Yaskawa INFORM job: R1_W43-44-A1(80,0))KM-OK.JBI

/JOB
//NAME R1_W43-44-A1(80,0))KM-OK
///FOLDERNAME KRIS-SCIANA
//POS
///NPOS 73,73,0,2,0,0
///TOOL 0
///POSTYPE PULSE
///PULSE
C00000=-135443,-162925,-128835,58859,85380,-57426
C00001=-92446,-155127,-126363,-9824,7934,-58174
C00002=-95529,-35335,-68837,19375,71902,-55615
C00003=-93187,-33344,-64604,18324,69907,-55135
C00004=-92721,-33324,-62151,18250,68383,-55215
C00005=-92468,-33122,-62017,18114,68351,-55131
C00006=-92880,-32499,-63991,18157,69897,-55031
C00007=-84694,-8010,-53588,6240,80947,-57198
C00008=-85014,-7064,-52060,6394,80518,-57316
C00009=-94295,-4530,-48038,22759,83190,-56081
C00010=-78802,-31555,-64347,-3071,67769,-50088
C00011=-78740,-31977,-64165,-3112,67443,-50058
C00012=-84933,-42926,-65553,8148,56142,-50726
C00013=-85694,-44675,-67677,8643,56621,-50981
C00014=-87687,-49011,-72903,9923,57813,-51634
C00015=-99004,-1535,-61632,22381,96772,-38436
C00016=-102646,2603,-65705,33052,95452,-62364
C00017=-97086,-22377,-78433,26069,74095,-68203
C00018=-96393,-22401,-76155,25819,72642,-68318
C00019=-97109,-22798,-76330,26266,72736,-68521
C00020=-97539,-22766,-76077,26544,72724,-68660
C00021=-97679,-22998,-75695,26674,72441,-68771
C00022=-99521,-21962,-80767,27350,76192,-68453
C00023=-70334,1557,-81441,-17401,103237,-40141
C00024=-67843,821,-73813,-18833,98965,-38392
C00025=-100316,3447,-64995,31985,94788,-61866
C00026=-99352,5668,-64520,31595,95249,-61456
C00027=-67843,821,-73813,-18833,98965,-38392
C00028=-85169,3045,-72107,6876,98019,-48310
C00029=-88969,4814,-69933,12844,98216,-50436
C00030=-98274,12123,-60045,27665,97638,-54760
C00031=-89932,6221,-75495,14866,97258,-51043
C00032=-93334,-9371,-63962,22562,99535,9595
C00033=-81626,10879,-49110,8622,108143,9572
C00034=-81231,10229,-48763,8499,107567,9646
C00035=-101964,-23029,-75036,41591,75550,70706
C00036=-102642,-26334,-76142,42122,75049,70241
C00037=-68700,15797,-43598,-6640,106638,27823
C00038=-63261,32591,-26999,-16022,110451,41229
C00039=-64996,36990,-21704,-15609,109207,40852
C00040=-64582,37586,-20939,-15664,109117,40995
C00041=-64496,38242,-20138,-15663,108980,41040
C00042=-64452,38361,-19695,-15647,108783,41080
C00043=-63126,40414,-20326,-16036,110391,41278
C00044=-63319,38327,-23499,-16110,111203,41105
C00045=-43516,29964,-10756,-46242,106248,64597
C00046=-43516,29964,-10756,-46242,106248,64597
C00047=-44396,28590,-11734,-46107,105755,64428
C00048=-43489,29718,-10008,-46103,105848,64806
C00049=-43472,27528,-13134,-46300,106419,64534
C00050=-43936,27041,-10805,-45843,105007,65003
C00051=-43522,29411,-9763,-46025,105613,64905
C00052=-42525,34492,-7112,-46386,106783,64798
C00053=-50383,13985,-41562,-28831,100075,68121
C00054=-64860,2482,-48793,-13393,87629,68164
C00055=-65930,5187,-46476,-12954,87445,67868
C00056=-57792,20564,-34513,-26464,97158,66415
C00057=-62898,8945,-45188,-24852,96370,64962
C00058=-63534,7410,-44996,-24591,95381,64971
C00059=-64227,9067,-43380,-24356,95073,64814
C00060=-63201,10906,-47674,-24936,98605,64395
C00061=-65206,-18847,-70813,-6241,82992,71232
C00062=-69426,-22420,-61359,-4258,75131,70311
C00063=-74955,-30598,-67106,-1464,74288,68599
C00064=-74021,-28518,-73716,-1903,79440,68812
C00065=-70812,-2884,-58486,-3475,83329,69650
C00066=-67265,-11111,-54966,-11415,75263,68927
C00067=-73959,-21777,-63314,-7907,74217,66930
C00068=-72807,-23542,-67362,-8463,75887,67172
C00069=-65188,-31999,-95671,-12172,89534,68158
C00070=-93091,-31999,-95671,-12172,89534,68158
C00071=-92446,-155127,-126363,-9824,7934,-58174
C00072=-92446,-155127,-126363,-9824,7934,84739
BC00000=21010,537295,1075111
BC00001=71,16,1075106
BC00002=15,15,1075175
BC00003=15,15,1075175
BC00004=15,15,1075175
BC00005=15,15,1075175
BC00006=15,15,1075175
BC00007=15,15,1075175
BC00008=15,15,1075175
BC00009=15,15,1075175
BC00010=15,15,1075175
BC00011=15,15,1075175
BC00012=15,15,1075175
BC00013=15,15,1075175
BC00014=15,15,1075175
BC00015=15,15,1006509
BC00016=15,15,928033
BC00017=15,15,898387
BC00018=15,15,898387
BC00019=15,15,898387
BC00020=15,15,898387
BC00021=15,15,898387
BC00022=15,15,898387
BC00023=15,15,898387
BC00024=15,15,898387
BC00025=15,15,901143
BC00026=15,15,901143
BC00027=15,15,898387
BC00028=15,15,898387
BC00029=15,15,898387
BC00030=15,15,898387
BC00031=15,15,898385
BC00032=15,15,1048834
BC00033=16,15,1047849
BC00034=16,15,1047849
BC00035=15,15,902068
BC00036=15,15,902068
BC00037=16,15,1047849
BC00038=16,16,1047846
BC00039=16,16,1047846
BC00040=16,16,1047846
BC00041=16,16,1047846
BC00042=16,16,1047846
BC00043=16,16,1047846
BC00044=16,16,1047846
BC00045=15,22410,1075175
BC00046=15,22410,1075175
BC00047=15,23652,1075175
BC00048=15,23652,1075175
BC00049=15,23652,1075175
BC00050=15,20488,1075175
BC00051=15,19247,1075175
BC00052=15,16142,1075175
BC00053=15,16142,1075175
BC00054=15,16142,1075175
BC00055=15,16142,1075175
BC00056=15,16142,1075175
BC00057=15,16142,1075175
BC00058=15,16142,1075175
BC00059=15,16142,1075175
BC00060=15,16142,1075175
BC00061=15,16142,1075173
BC00062=15,16142,1075173
BC00063=15,16142,1075173
BC00064=15,16142,1075173
BC00065=15,16142,1075173
BC00066=15,16142,1075173
BC00067=15,16142,1075173
BC00068=15,16142,1075173
BC00069=15,16142,1075173
BC00070=15,16142,1075173
BC00071=71,16,1075106
BC00072=388530,120,1075106
///POSTYPE BASE
///RECTAN
///RCONF 0,0,0,0,1,0,0,0,0,0,0,0,0,0,0,0,0,0,0,0,0,0,0,0
P00006=2.006,1.622,-0.565,0.0000,0.0000,0.0000
///RCONF 0,0,0,0,0,0,0,0,0,0,0,0,0,0,0,0,0,0,0,0,0,0,0,0
P00023=-2.957,-4.083,2.762,0.0000,0.0000,0.0000
//INST
///DATE 2024/09/16 12:17
///ATTR SC,RW
///GROUP1 RB1,BS1
NOP
'r1_W43-44-A1(80,0))
'Path S1224
MOVJ C00000 BC00000 VJ=100.00
MOVJ C00001 BC00001 VJ=100.00
SFTOF
MOVJ C00002 BC00002 VJ=100.00
MOVJ C00003 BC00003 VJ=100.00
MOVL C00004 BC00004 V=60.0
REFP 3 C00005 BC00005
CALL JOB:SEARCH-R1
SET P023 P006
SFTON P023
MOVL C00006 BC00006 V=60.0
MOVL C00007 BC00007 V=60.0
REFP 3 C00008 BC00008
CALL JOB:SEARCH-R1
SET P023 P006
SFTON P023
MOVL C00009 BC00009 V=60.0
MOVL C00010 BC00010 V=60.0
REFP 3 C00011 BC00011
CALL JOB:SEARCH-R1
SET P023 P006
SFTON P023
MOVL C00012 BC00012 V=60.0
MOVL C00013 BC00013 V=166.7
MOVL C00014 BC00014 V=166.7
'Path VIA1253
SFTOF
CALL JOB:COFNIJ_DRUT
MOVJ C00015 BC00015 VJ=100.00
'Path W1225
SFTOF
SFTON P023
MOVJ C00016 BC00016 VJ=100.00
MACRO1 MJ#(0) ARGF7
MOVJ C00017 BC00017 VJ=100.00
MOVJ C00018 BC00018 VJ=100.00
ARCON
MOVL C00019 BC00019 V=8.3
MOVL C00020 BC00020 V=8.3
MOVL C00021 BC00021 V=8.3
ARCOF
MOVJ C00022 BC00022 VJ=15.00
MOVJ C00023 BC00023 VJ=100.00
MOVL C00024 BC00024 V=100.0 PL=0
REFP 1 C00025 BC00025
REFP 2 C00026 BC00026
MACRO1 MJ#(0) ARGF7
ARCON
MOVL C00027 BC00027 V=10.0
MOVL C00028 BC00028 V=10.0
MOVL C00029 BC00029 V=10.0
MOVL C00030 BC00030 V=10.0
ARCOF
MOVL C00031 BC00031 V=166.7
MOVL C00032 BC00032 V=166.7
'Path W1226
SFTOF
SFTON P023
MOVJ C00033 BC00033 VJ=100.00
MOVL C00034 BC00034 V=100.0 PL=0
REFP 1 C00035 BC00035
REFP 2 C00036 BC00036
MACRO1 MJ#(0) ARGF7
ARCON
MOVL C00037 BC00037 V=10.0
MOVL C00038 BC00038 V=10.0
MOVL C00039 BC00039 V=10.0
MACRO1 MJ#(0) ARGF7
MOVL C00040 BC00040 V=8.3
MOVL C00041 BC00041 V=8.3
MOVL C00042 BC00042 V=8.3
ARCOF
MOVL C00043 BC00043 V=166.7
MOVL C00044 BC00044 V=166.7
SFTOF
'Path VIA1252
SFTON P023
MOVJ C00045 BC00045 VJ=100.00
SFTOF
SFTON P023
MOVJ C00046 BC00046 VJ=100.00
MOVL C00047 BC00047 V=100.0 PL=0
REFP 1 C00048 BC00048
REFP 2 C00049 BC00049
MACRO1 MJ#(0) ARGF9
ARCON
MOVL C00050 BC00050 V=10.0
ARCOF
MOVL C00051 BC00051 V=166.7
MOVL C00052 BC00052 V=166.7
SFTOF
MOVJ C00053 BC00053 VJ=100.00
MACRO1 MJ#(0) ARGF6
MOVJ C00054 BC00054 VJ=100.00
'ARCON
MOVL C00055 BC00055 V=8.3
'ARCOFF
MOVJ C00056 BC00056 VJ=100.00
MOVJ C00057 BC00057 VJ=100.00
MOVJ C00058 BC00058 VJ=100.00
'ARCON
MOVL C00059 BC00059 V=9.2
'ARCOFF
MOVJ C00060 BC00060 VJ=100.00
MOVJ C00061 BC00061 VJ=100.00
MOVJ C00062 BC00062 VJ=100.00
ARCON
TIMER T=0.50
ARCOF
MOVJ C00063 BC00063 VJ=100.00
ARCON
TIMER T=0.50
ARCOF
MOVJ C00064 BC00064 VJ=100.00
MOVJ C00065 BC00065 VJ=100.00
MACRO1 MJ#(0) ARGF7
MOVJ C00066 BC00066 VJ=100.00
ARCON
MOVL C00067 BC00067 V=7.5
ARCOF
MOVJ C00068 BC00068 VJ=20.00
MOVJ C00069 BC00069 VJ=100.00
MOVJ C00070 BC00070 VJ=100.00
MOVJ C00071 BC00071 VJ=100.00
MOVJ C00072 BC00072 VJ=100.00
SFTOF
END
